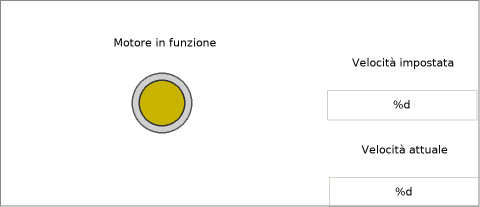
VISUALIZATION Visualization  // 480x207
    Lamp1 (127,68 70x70), variable: GVL_SA.singleAxis.Status.Moving, style: Lamp-Lamp1-Yellow
    Textfield (327,90 150x30), "%d", text variable: GVL_SA.stSA_VelCmd1.lrVelocity
    Label (328,48 150x30), "Velocità impostata"
    Label (90,28 150x30), "Motore in funzione"
    Textfield (329,177 150x30), "%d", text variable: GVL_SA.singleAxis.NcToPlc.ActVelo
    Label (330,135 150x30), "Velocità attuale"
END_VISUALIZATION

(* stored: Version 1.1.0.1, ProductVersion 3.1.4024.12
   Visu Visualization: Id {81299271-388a-4b91-956a-6f6401640dca} *)
